TYPE ST_CylinderParCmd :
STRUCT
    Reserved : BOOL;
END_STRUCT
END_TYPE

(* stored: Version 1.1.0.1, ProductVersion 3.1.4024.12
   DUT ST_CylinderParCmd: Id {9e72dc72-3935-49dd-a778-319a057cf2af} *)
